INTERFACE I_TankController

METHOD ApplyCooling 
VAR_INPUT
END_VAR
END_METHOD

METHOD CheckSafety
VAR_INPUT
END_VAR
END_METHOD

METHOD DispenseChemical 
VAR_INPUT
END_VAR
END_METHOD

END_INTERFACE

(* stored: Version 1.1.0.1, ProductVersion 3.1.4024.16
   Itf I_TankController: Id {d87c8149-f9f5-4fdf-9ce3-1e9e03dcebc9}
   Method ApplyCooling: Id {d010dc96-5077-445e-9fd3-273069478e21}
   Method CheckSafety: Id {822e6ffb-3777-4f38-b443-13017b990ca7}
   Method DispenseChemical: Id {3a6fd6f1-e5b7-4545-96d4-3892704c8127} *)
